Fanuc KAREL source: kd00076.KL

-- PROVISIONAL review KL for V940-1; original PC SHA256 d215d2a85d7efa43b1a674d575f39f06f676e9c3d157d561d5c1aea86ac8c740
-- Incomplete behavior may be omitted. Consult companion uncertainty JSON. Do not deploy.
PROGRAM KD00076
%NOLOCKGROUP
VAR
  I : INTEGER
  J : INTEGER
  B : BOOLEAN
  R : REAL
  S : STRING[80]
BEGIN
  -- V9_ZERO_TABLE_METADATA_HINT layout=0001; no indexed target words; source/name/runtime held
  -- UNRESOLVED_PC offsets 5-7; opcodes 9D,3C
  -- UNRESOLVED_PC offsets 12-16; opcodes 7F
END KD00076
